// TwinCAT 3 PLC project
// project tree:
//   POUs/ func_f1.TcPOU, func_f2.TcPOU, func_fac.TcPOU, ifExprFunc1.TcPOU, func_fac2.TcPOU, func_fac3.TcPOU, alg_g_algeb1.TcPOU, makeTupleStruct_1.TcPOU, proj0_TupleStruct_1.TcPOU (not stored), proj1_TupleStruct_1.TcPOU, alg_g_algeb2.TcPOU, makeTupleStruct_2.TcPOU, proj0_TupleStruct_2.TcPOU, proj1_TupleStruct_2.TcPOU, makeTupleStruct_3.TcPOU, proj0_TupleStruct_3.TcPOU, proj1_TupleStruct_3.TcPOU, derivcvar_M_p_t.TcPOU (not stored), derivcvar_M_p_t2.TcPOU, derivcvar_M_p_t3.TcPOU, MAIN.TcPOU
//   DUTs/ STATE.TcDUT, enum_E.TcDUT, TupleStruct_1.TcDUT, TupleStruct_2.TcDUT, TupleStruct_3.TcDUT
//   GVLs/ INPUTS.TcGVL, TIMERS.TcGVL (not stored)

// ---- DUTs/STATE.TcDUT
TYPE STATE:
    STRUCT
        curTime: LREAL;
        dvar_M_p_b AT %Q*: BOOL;
        dvar_M_p_x AT %Q*: DINT;
        dvar_M_p_y AT %Q*: LREAL;
        dvar_M_p_ve AT %Q*: enum_E;
        dvar_M_p_v1 AT %Q*: DINT;
        dvar_M_p_v2 AT %Q*: TupleStruct_1;
        dvar_M_p_v3 AT %Q*: TupleStruct_2;
        dvar_M_p_tv AT %Q*: TupleStruct_3;
        dvar_M_p_j AT %Q*: DINT;
        dvar_M_p_r AT %Q*: LREAL;
        cvar_M_p_t AT %Q*: LREAL;
        cvar_M_p_t2 AT %Q*: LREAL;
        cvar_M_p_t3 AT %Q*: LREAL;
        dvar_M_p AT %Q*: enum_E;
    END_STRUCT
END_TYPE

// ---- DUTs/enum_E.TcDUT
TYPE enum_E:
    (elit_l1, elit_l10, elit_l11, elit_l12, elit_l13, elit_l14, elit_l15, elit_l16, elit_l2, elit_l3, elit_l4, elit_l5, elit_l6, elit_l7, elit_l8, elit_l9, elit_LIT1, elit_LIT2);
END_TYPE

// ---- DUTs/TupleStruct_1.TcDUT
TYPE TupleStruct_1:
    STRUCT
        field0: LREAL;
        field1: LREAL;
    END_STRUCT
END_TYPE

// ---- DUTs/TupleStruct_2.TcDUT
TYPE TupleStruct_2:
    STRUCT
        field0: TupleStruct_1;
        field1: LREAL;
    END_STRUCT
END_TYPE

// ---- DUTs/TupleStruct_3.TcDUT
TYPE TupleStruct_3:
    STRUCT
        field0: DINT;
        field1: DINT;
    END_STRUCT
END_TYPE

// ---- GVLs/INPUTS.TcGVL
VAR_GLOBAL // INPUTS
    ivar_g_inp AT %I*: DINT;
END_VAR

// ---- POUs/func_f1.TcPOU
FUNCTION func_f1: DINT
VAR_INPUT
    farg_f1_x: DINT;
END_VAR

func_f1 := (farg_f1_x) + (1);
RETURN;

END_FUNCTION

// ---- POUs/func_f2.TcPOU
FUNCTION func_f2: LREAL
VAR_INPUT
    farg_f2_y: LREAL;
END_VAR
VAR
    fvar_f2_z: LREAL;
END_VAR

// Initialize local variables.
fvar_f2_z := farg_f2_y;

// Actual function body.
IF ((farg_f2_y) > (0)) THEN
    func_f2 := fvar_f2_z;
    RETURN;
ELSE
    func_f2 := (fvar_f2_z) + (1.0);
    RETURN;
END_IF;

END_FUNCTION

// ---- POUs/func_fac.TcPOU
FUNCTION func_fac: DINT
VAR_INPUT
    farg_fac_a: DINT;
END_VAR

func_fac := ifExprFunc1(farg_fac_a);
RETURN;

END_FUNCTION

// ---- POUs/ifExprFunc1.TcPOU
FUNCTION ifExprFunc1: DINT
VAR_INPUT
    farg_fac_a: DINT;
END_VAR

IF ((farg_fac_a) = (0)) THEN
    ifExprFunc1 := 1;
ELSE
    ifExprFunc1 := (func_fac((farg_fac_a) - (1))) * (farg_fac_a);
END_IF;

END_FUNCTION

// ---- POUs/func_fac2.TcPOU
FUNCTION func_fac2: DINT
VAR_INPUT
    farg2_fac2_a: DINT;
END_VAR
VAR
    farg_fac2_a: DINT;
    fvar_fac2_rslt: DINT;
END_VAR

farg_fac2_a := farg2_fac2_a;
// Initialize local variables.
fvar_fac2_rslt := 1;

// Actual function body.
WHILE ((farg_fac2_a) > (0)) DO
    fvar_fac2_rslt := (fvar_fac2_rslt) * (farg_fac2_a);
    farg_fac2_a := (farg_fac2_a) - (1);
END_WHILE;
func_fac2 := fvar_fac2_rslt;
RETURN;

END_FUNCTION

// ---- POUs/func_fac3.TcPOU
FUNCTION func_fac3: DINT
VAR_INPUT
    farg2_fac3_a: DINT;
END_VAR
VAR
    farg_fac3_a: DINT;
    fvar_fac3_rslt: DINT;
END_VAR

farg_fac3_a := farg2_fac3_a;
// Initialize local variables.
fvar_fac3_rslt := 1;

// Actual function body.
WHILE (TRUE) DO
    IF ((farg_fac3_a) < (1)) THEN
        EXIT;
    END_IF;
    fvar_fac3_rslt := (fvar_fac3_rslt) * (farg_fac3_a);
    farg_fac3_a := (farg_fac3_a) - (1);
END_WHILE;
func_fac3 := fvar_fac3_rslt;
RETURN;

END_FUNCTION

// ---- POUs/alg_g_algeb1.TcPOU
FUNCTION alg_g_algeb1: LREAL
VAR_INPUT
    state: STATE;
END_VAR

alg_g_algeb1 := (state.curTime) + (1.0);

END_FUNCTION

// ---- POUs/makeTupleStruct_1.TcPOU
FUNCTION makeTupleStruct_1: TupleStruct_1
VAR_INPUT
    field0: LREAL;
    field1: LREAL;
END_VAR
VAR
    rslt: TupleStruct_1;
END_VAR

rslt.field0 := field0;
rslt.field1 := field1;
makeTupleStruct_1 := rslt;

END_FUNCTION

// ---- POUs/proj1_TupleStruct_1.TcPOU

      FUNCTION proj1_TupleStruct_1: LREAL
VAR_INPUT
    tuple: TupleStruct_1;
END_VAR


        proj1_TupleStruct_1 := tuple.field1;

END_FUNCTION

// ---- POUs/alg_g_algeb2.TcPOU
FUNCTION alg_g_algeb2: TupleStruct_1
VAR_INPUT
    state: STATE;
END_VAR

alg_g_algeb2 := makeTupleStruct_1(state.curTime, (state.curTime) + (1.0));

END_FUNCTION

// ---- POUs/makeTupleStruct_2.TcPOU
FUNCTION makeTupleStruct_2: TupleStruct_2
VAR_INPUT
    field0: TupleStruct_1;
    field1: LREAL;
END_VAR
VAR
    rslt: TupleStruct_2;
END_VAR

rslt.field0 := field0;
rslt.field1 := field1;
makeTupleStruct_2 := rslt;

END_FUNCTION

// ---- POUs/proj0_TupleStruct_2.TcPOU
FUNCTION proj0_TupleStruct_2: TupleStruct_1
VAR_INPUT
    tuple: TupleStruct_2;
END_VAR

proj0_TupleStruct_2 := tuple.field0;

END_FUNCTION

// ---- POUs/proj1_TupleStruct_2.TcPOU
FUNCTION proj1_TupleStruct_2: LREAL
VAR_INPUT
    tuple: TupleStruct_2;
END_VAR

proj1_TupleStruct_2 := tuple.field1;

END_FUNCTION

// ---- POUs/makeTupleStruct_3.TcPOU
FUNCTION makeTupleStruct_3: TupleStruct_3
VAR_INPUT
    field0: DINT;
    field1: DINT;
END_VAR
VAR
    rslt: TupleStruct_3;
END_VAR

rslt.field0 := field0;
rslt.field1 := field1;
makeTupleStruct_3 := rslt;

END_FUNCTION

// ---- POUs/proj0_TupleStruct_3.TcPOU
FUNCTION proj0_TupleStruct_3: DINT
VAR_INPUT
    tuple: TupleStruct_3;
END_VAR

proj0_TupleStruct_3 := tuple.field0;

END_FUNCTION

// ---- POUs/proj1_TupleStruct_3.TcPOU
FUNCTION proj1_TupleStruct_3: DINT
VAR_INPUT
    tuple: TupleStruct_3;
END_VAR

proj1_TupleStruct_3 := tuple.field1;

END_FUNCTION

// ---- POUs/derivcvar_M_p_t2.TcPOU
FUNCTION derivcvar_M_p_t2: LREAL
VAR_INPUT
    state: STATE;
END_VAR

derivcvar_M_p_t2 := 2.0;

END_FUNCTION

// ---- POUs/derivcvar_M_p_t3.TcPOU
FUNCTION derivcvar_M_p_t3: LREAL
VAR_INPUT
    state: STATE;
END_VAR

derivcvar_M_p_t3 := state.cvar_M_p_t3;

END_FUNCTION

// ---- POUs/MAIN.TcPOU
PROGRAM MAIN
VAR_OUTPUT
    timerValue0: TIME;
    timerValue1: TIME;
END_VAR
VAR
    cnt: LINT;
    first: BOOL := TRUE;
    curTimerValue: TIME;
    state0: STATE;
    curTime: LREAL;
    loopsKilled: LINT;
END_VAR
VAR_TEMP
    lastTimerValue: TIME;
    curDeltaTime: TIME;
    curDeltaSecs: LREAL;
    state1: STATE;
    progress: BOOL;
    loopCount: INT;
END_VAR


// Handle 'time' and cycle time.
cnt := cnt + 1;

timer0(IN := curTimer = 0, PT := T#1D);
timer1(IN := curTimer = 1, PT := T#1D);
timerValue0 := timer0.ET;
timerValue1 := timer1.ET;

lastTimerValue := curTimerValue;
IF curTimer = 0 THEN
    curTimerValue := timerValue0;
ELSE
    curTimerValue := timerValue1;
END_IF;
curDeltaTime := curTimerValue - lastTimerValue;
curDeltaSecs := TIME_TO_LREAL(curDeltaTime) / 1000;
curTime := curTime + curDeltaSecs;

IF cnt MOD 10 = 0 THEN
    curTimer := 1 - curTimer;
    curTimerValue := T#0S;
    timer0(IN := curTimer = 0, PT := T#1D);
    timer1(IN := curTimer = 1, PT := T#1D);
    timerValue0 := timer0.ET;
    timerValue1 := timer1.ET;
END_IF;

IF first THEN
    first := FALSE;

    // Initialize state variables for initial state.
    state0.dvar_M_p_b := TRUE;
    state0.dvar_M_p_x := 0;
    state0.dvar_M_p_y := 1.23;
    state0.dvar_M_p_ve := elit_LIT1;
    state0.dvar_M_p_v1 := 0;
    state0.dvar_M_p_v2 := makeTupleStruct_1(0.0, 0.0);
    state0.dvar_M_p_v3 := makeTupleStruct_2(makeTupleStruct_1(0.0, 0.0), 0.0);
    state0.dvar_M_p_tv := makeTupleStruct_3(0, 0);
    state0.dvar_M_p_j := 0;
    state0.dvar_M_p_r := 1000000.0;
    state0.cvar_M_p_t := 0.0;
    state0.cvar_M_p_t2 := 1.0;
    state0.cvar_M_p_t3 := 0.0;
    state0.dvar_M_p := elit_l1;
ELSE
    // Update continuous variables for time delay.
    state1.cvar_M_p_t := state0.cvar_M_p_t + curDeltaSecs * derivcvar_M_p_t(state0);
    state1.cvar_M_p_t2 := state0.cvar_M_p_t2 + curDeltaSecs * derivcvar_M_p_t2(state0);
    state1.cvar_M_p_t3 := state0.cvar_M_p_t3 + curDeltaSecs * derivcvar_M_p_t3(state0);

    state0.curTime := curTime;
    state0.cvar_M_p_t := state1.cvar_M_p_t;
    state0.cvar_M_p_t2 := state1.cvar_M_p_t2;
    state0.cvar_M_p_t3 := state1.cvar_M_p_t3;
END_IF;

// Event loop.
WHILE TRUE DO
    progress := FALSE;

    // Event "tau".
    IF NOT progress THEN
        IF (state0.dvar_M_p) = (elit_l1) THEN
            progress := TRUE;
            state1 := state0;

            state1.dvar_M_p_v1 := func_f1(state0.dvar_M_p_x);
            state1.dvar_M_p := elit_l2;

            state0 := state1;
        END_IF;
    END_IF;

    // Event "tau".
    IF NOT progress THEN
        IF (state0.dvar_M_p) = (elit_l2) THEN
            progress := TRUE;
            state1 := state0;

            state1.dvar_M_p_v2 := alg_g_algeb2(state0);
            state1.dvar_M_p := elit_l3;

            state0 := state1;
        END_IF;
    END_IF;

    // Event "tau".
    IF NOT progress THEN
        IF (state0.dvar_M_p) = (elit_l3) THEN
            progress := TRUE;
            state1 := state0;

            state1.dvar_M_p_y := (func_f2(0.0)) + (func_f2(state0.dvar_M_p_y));
            state1.dvar_M_p := elit_l4;

            state0 := state1;
        END_IF;
    END_IF;

    // Event "tau".
    IF NOT progress THEN
        IF (state0.dvar_M_p) = (elit_l4) THEN
            progress := TRUE;
            state1 := state0;

            state1.dvar_M_p_x := ((func_fac(4)) + (func_fac2(4))) + (func_fac3(4));
            state1.dvar_M_p := elit_l5;

            state0 := state1;
        END_IF;
    END_IF;

    // Event "tau".
    IF NOT progress THEN
        IF (state0.dvar_M_p) = (elit_l5) THEN
            progress := TRUE;
            state1 := state0;

            state1.dvar_M_p_tv := makeTupleStruct_3(1, 2);
            state1.dvar_M_p := elit_l6;

            state0 := state1;
        END_IF;
    END_IF;

    // Event "tau".
    IF NOT progress THEN
        IF (state0.dvar_M_p) = (elit_l6) THEN
            progress := TRUE;
            state1 := state0;

            state1.dvar_M_p_x := proj0_TupleStruct_3(makeTupleStruct_3(3, 4));
            state1.dvar_M_p_j := proj1_TupleStruct_3(makeTupleStruct_3(3, 4));
            state1.dvar_M_p := elit_l7;

            state0 := state1;
        END_IF;
    END_IF;

    // Event "tau".
    IF NOT progress THEN
        IF (state0.dvar_M_p) = (elit_l7) THEN
            progress := TRUE;
            state1 := state0;

            state1.dvar_M_p_x := proj0_TupleStruct_3(state0.dvar_M_p_tv);
            state1.dvar_M_p_j := proj1_TupleStruct_3(state0.dvar_M_p_tv);
            state1.dvar_M_p := elit_l8;

            state0 := state1;
        END_IF;
    END_IF;

    // Event "tau".
    IF NOT progress THEN
        IF (state0.dvar_M_p) = (elit_l8) THEN
            progress := TRUE;
            state1 := state0;

            state1.dvar_M_p_tv.field0 := 5;
            state1.dvar_M_p := elit_l9;

            state0 := state1;
        END_IF;
    END_IF;

    // Event "tau".
    IF NOT progress THEN
        IF (state0.dvar_M_p) = (elit_l9) THEN
            progress := TRUE;
            state1 := state0;

            state1.dvar_M_p_tv.field1 := proj0_TupleStruct_3(makeTupleStruct_3(6, 7));
            state1.dvar_M_p_j := proj1_TupleStruct_3(makeTupleStruct_3(6, 7));
            state1.dvar_M_p := elit_l10;

            state0 := state1;
        END_IF;
    END_IF;

    // Event "tau".
    IF NOT progress THEN
        IF (state0.dvar_M_p) = (elit_l10) THEN
            progress := TRUE;
            state1 := state0;

            state1.dvar_M_p_v3.field0.field1 := 7.8;
            state1.dvar_M_p := elit_l11;

            state0 := state1;
        END_IF;
    END_IF;

    // Event "tau".
    IF NOT progress THEN
        IF (state0.dvar_M_p) = (elit_l11) THEN
            progress := TRUE;
            state1 := state0;

            state1.dvar_M_p_v3 := makeTupleStruct_2(makeTupleStruct_1(1.2, 3.4), 5.6);
            state1.dvar_M_p := elit_l12;

            state0 := state1;
        END_IF;
    END_IF;

    // Event "tau".
    IF NOT progress THEN
        IF (state0.dvar_M_p) = (elit_l12) THEN
            progress := TRUE;
            state1 := state0;

            state1.dvar_M_p_j := (state0.dvar_M_p_j) + (1);
            state1.dvar_M_p := elit_l13;

            state0 := state1;
        END_IF;
    END_IF;

    // Event "tau".
    IF NOT progress THEN
        IF (state0.dvar_M_p) = (elit_l13) THEN
            progress := TRUE;
            state1 := state0;

            state1.dvar_M_p_b := FALSE;
            state1.dvar_M_p := elit_l14;

            state0 := state1;
        END_IF;
    END_IF;

    // Event "tau".
    IF NOT progress THEN
        IF (state0.dvar_M_p) = (elit_l14) THEN
            progress := TRUE;
            state1 := state0;

            IF (NOT(state0.dvar_M_p_b)) THEN
                state1.dvar_M_p_ve := elit_LIT2;
            END_IF;
            state1.dvar_M_p := elit_l15;

            state0 := state1;
        END_IF;
    END_IF;

    // Event "tau".
    IF NOT progress THEN
        IF (state0.dvar_M_p) = (elit_l15) THEN
            progress := TRUE;
            state1 := state0;

            state1.dvar_M_p_r := (ivar_g_inp) + (10.0);
            state1.dvar_M_p := elit_l16;

            state0 := state1;
        END_IF;
    END_IF;

    // Done with events?
    IF NOT progress THEN
        EXIT;
    END_IF;

    // Protect against events that are always enabled.
    loopCount := loopCount + 1;
    IF loopCount >= 100 THEN
        loopsKilled := loopsKilled + 1;
        EXIT;
    END_IF;
END_WHILE;

END_PROGRAM
